(* IEC 61131-3 sources: verifaps-lib/geteta/examples/issue1, 1 file *)

(* ---- issue1.st ---- *)
PROGRAM constantprogram
  VAR_INPUT
    A : INT;
    B : BOOL;
  END_VAR

  VAR_OUTPUT
    C : INT;
    D : BOOL;
  END_VAR

  C := 52;
END_PROGRAM
